PROGRAM MAIN
VAR
    sVersion: STRING:='1.0.0';
    i : UINT; //index variable for AXES()
    aFbAxes: ARRAY [1..gvl_app.axisNum] OF FB_Axis;
    hmiAxisSelection    :   INT:=1;     //Not possible to use local hmi variables for array indexes

(******Outputs: Power for Limit switches and Home Sensors (every 4th output)********)

    bOutput1 AT %Q*: BOOL:= TRUE;
    //bOutput2 AT %Q*: BOOL:= TRUE;
    //bOutput3 AT %Q*: BOOL:= TRUE;
    //bOutput4 AT %Q*: BOOL:= TRUE;
    //bOutput5 AT %Q*: BOOL:= TRUE;
    //bOutput6 AT %Q*: BOOL:= TRUE;
    //bOutput7 AT %Q*: BOOL:= TRUE;
    //bOutput8 AT %Q*: BOOL:= TRUE;
    //bOutput9 AT %Q*: BOOL:= TRUE;
    //bOutput13 AT %Q*: BOOL:= TRUE;
    //bOutput17 AT %Q*: BOOL:= TRUE;
    //bOutput21 AT %Q*: BOOL:= TRUE;
    //bOutput24 AT %Q*: BOOL:= TRUE;
    //bOutput28 AT %Q*: BOOL:= TRUE;

(******Error Handling********)
    fbErrorSystem: FB_ErrorSystem;
    aFbAxesError: ARRAY [1..gvl_app.axisNum] OF FB_NC_Error;

    //fbEL1018  : EL1018;
    //fbEL2808  : EL2808;
    //fbEL5101  : EL5101;
    //fbEL9505  : EL9505;
    //fbEL1252  : EL1252;
    //fbEL9410  : EL9410;
    //fbEL7037  : EL7037;
    //fbEK1110  : EK1110;

(******Startup, Shutdown and UPS********)
    fbUPS                  : FB_S_UPS_CX51x0;
    eUpsMode               : E_S_UPS_Mode   := eSUPS_WrPersistData_Shutdown;
    eStartUp: (ColdStart, ReadAxisFeedbackType, CheckReadDone, ExecuteRestore, CheckRestore, FinishRestore);
    bPositionRestoreDone   : BOOL := FALSE;
    bRestoreExecute        : BOOL := FALSE;
    bExecuteReadEncRefSys  : BOOL := FALSE;
    iRetry                 : INT;
    fbReadEncRefSys        : ARRAY [1..gvl_app.axisNum] OF MC_ReadParameter;
    fbRestorePosition      : ARRAY [1..GVL_app.axisNum] OF MC_SetPosition;

END_VAR

VAR PERSISTENT
    bRestoreOnStartup : BOOL;
END_VAR

fbUPS(eUpsMode := eUpsMode); (* call UPS-FB instance in first lines of the fastest PLC Task *)

IF eGlobalSUpsState = eSUPS_PowerFailure THEN
    (* first cycle of powerfailure *)
    (* execute code that should only be done once with each powerfailure, i.e. increase powerfailure counter *)
    bRestoreOnStartup:=TRUE;
    STORE_PERSISTENT();
    RETURN;
ELSIF eGlobalSUpsState > eSUPS_PowerFailure THEN
    (* next cycles of powerfailure *)
    (* skip regular code execution for the remaining cycles of the powerfailure/writing of persistent data/quick shutdown  ... *)
    RETURN;
END_IF

RESTORE_POSITIONS();
PROG();
AXES();
ERROR();

ACTION AXES:
FOR GVL.iAxis:=1 TO gvl_app.axisNum DO
    aFbAxes[GVL.iAxis](stAxisStruct:=gvl.axes[GVL.iAxis]);
END_FOR
END_ACTION

ACTION ERROR:
//
(****FB containting the log of the errors****)
//
fbErrorSystem(
    En:= TRUE,
    bReset:= ,
    nErrorNum:= ,
    bACK:= ,
    bValidSelection:= ,
    nTableRowIndex:= ,
    EnO=> ,
    nSelectedError=> ,
    pErrorSystem=> );


FOR GVL.iAxis:=1 TO gvl_app.axisNum DO
    aFbAxesError[gvl.iAxis](EN:=TRUE,
    nNC_ErrorID:= gvl.axes[gvl.iAxis].status.nErrorID,
    nNC_AxisID:=gvl.axes[gvl.iAxis].Axis.NcToPlc.AxisId,
    ErrorSystem:= fbErrorSystem.pErrorSystem);
END_FOR



(*call all the necessary instance (input assistance F2 or right click) according to the terminals that you have in your hardware and
 add "TRUE" in the input En, the corresponding number of termianl to the iTerminal_ID and
the variable "fbErrorSystem.pErrorSystem" to the input ErrorSystem in each FB E. g. :
fbEL1808(
    En:= TRUE,
    iTerminal_ID:= 01,
    ErrorSystem:= fbErorSystem.pErrorSystem,
    EnO=> ,
    bError=> );
 *)
END_ACTION

ACTION PROG:
//
(* Program any sequence, safety or feature (if necessary) application specific in thsi section*)

//
END_ACTION

ACTION RESTORE_POSITIONS:
///#########################################################
// This ACT will restore the position of an incremental axis on startup with the act position it read before losing power.
// It checks the type of axis, 0=incremental, and that the axis was stationary at shut down.
// Because 0 equates to incremental we also need to check that the data is valid, otherwise by default it would restore all axes.
// By default an axis will not restore the position unless it is set to opt-in, i.e. gvl.axes[i].config.eRestorePosition is non-zero.
// This needs to be initialised somewhere in TwinCAT code otherwise it will not be available at start up.
// A restore will only be performed on a loss of power, this code shouldn't make any changes on a reset cold, a rest origin or a download.
// There is a enum to allow for different types of restore modes, currently only one is implemented.
// 0 'DontRestore'
// 1 'RestoreWithoutHome' -restores the position using a set position fb and does not set the home bit in the axis struct.
// Note from Beckhoff: "A maximum of 1 MB persistent data can be reliably saved over the entire service life."
///#########################################################

IF bRestoreOnStartup THEN
    bRestoreOnStartup:=FALSE;
    bRestoreExecute:=TRUE;
END_IF

// Upon startup bPositionRestoreDone will be set to FALSE, after successfully completing the following code it will be set TRUE
// and should stay TRUE for the rest of the time the PLC is operational, thus this routine should only be completed once.
IF bRestoreExecute AND NOT bPositionRestoreDone THEN

    // Cycle through function blocks that read the encoder reference system i.e. whether axis is incremental or absolute
    // Result stored in Value, 0=Inc 1=Abs, execute set during the case statement
    FOR i:=1 TO gvl_app.axisNum DO
        fbReadEncRefSys[i](
          Axis:= gvl.axes[i].Axis,
          Enable:= bExecuteReadEncRefSys,
          ParameterNumber:= MC_AxisParameter.AxisEncoderReferenceSystem,
          Value=>,
          ReadMode:= E_READMODE.READMODE_ONCE);
    END_FOR

    // Cycle through set position function blocks for each axis
    FOR i:=1 TO gvl_app.axisNum DO
        fbRestorePosition[i](
         Axis:= gvl.axes[i].Axis,
         Execute:= ,
         Position:= axesPersistent[i].iPositionAtShutdown);
    END_FOR

    CASE eStartUp OF
        ColdStart:
        // First cycle of the PLC, do nothing just give one cycle for variables to initialise
            IF NOT bPositionRestoreDone THEN
                eStartUp:=eStartUp+1;
                iRetry:=0;
            END_IF

        ReadAxisFeedbackType:
        // Exectute the function blocks to read the encoder reference system (0=inc OR 1=ABS)
            bExecuteReadEncRefSys:=TRUE;
            eStartUp:=eStartUp+1;

        CheckReadDone:
        // Check the encoder reference system has been read for all axis -> if busy then continue with PLC cycle and check again next time.
        // If fbReadEncRefSys not started then go back a step.
        // If any axes result in an error the code will get stuck here, this happens if gvl_app.axisNum is not set correctly
            FOR i:=1 TO gvl_app.axisNum DO
                IF fbReadEncRefSys[i].Valid = FALSE THEN
                    IF fbReadEncRefSys[i].Busy = TRUE THEN
                        // Exit MAIN.STARTUP Action and wait till next cycle, needs to cycle through whole program in order for data to update
                        RETURN;
                    ELSE
                        // Sometimes the code gets here and the fbReadEncRefSys[i] misses the rising edge. If  the code gets here it means
                        // .valid=FALSE and .busy=FALSE which indicateds the FB probably hasn't started and thus needs to see a rising edge.
                        // Set execute to low, Exit MAIN.STARTUP and go back a step in the CASE statement.
                        bExecuteReadEncRefSys:=FALSE;
                        eStartUp:=eStartUp-1;
                        iRetry:=iRetry+1; // counter used for troubleshooting to see how many cycles it takes before fbReadEncRefSys function blocks are read correctly
                        RETURN;
                    END_IF
                END_IF
            END_FOR
            // If the code gets here all axes either have .valid=TRUE for all axes
            eStartUp:=eStartUp+1;

        ExecuteRestore:
        // Execute position restore by setting fbRestorePosition.execute = TRUE
            FOR i:=1 TO gvl_app.axisNum DO
                IF fbReadEncRefSys[i].Valid = TRUE AND fbReadEncRefSys[i].Value = 0 AND NOT(axesPersistent[i].bMovingAtShutdown) THEN
                    IF GVL.axes[i].config.eRestorePosition = RestorePosition.RestoreWithoutHome THEN
                        fbRestorePosition[i].Execute:=TRUE;
                    END_IF
                END_IF
            END_FOR
            eStartUp:=eStartUp+1;

        CheckRestore:
        // Check the set position fbs are finished
        // Nothing actually happens if the restore is not done, the code just returns from here each cycle and the
        // bPositionRestoreDone will never get set to TRUE and will take up cycle time
            FOR i:=1 TO gvl_app.axisNum DO
                IF fbReadEncRefSys[i].Valid = TRUE AND fbReadEncRefSys[i].Value = 0 AND NOT(axesPersistent[i].bMovingAtShutdown) THEN
                    IF GVL.axes[i].config.eRestorePosition = RestorePosition.RestoreWithoutHome THEN
                        IF NOT fbRestorePosition[i].Done THEN
                            RETURN;
                        END_IF
                    END_IF
                END_IF
            END_FOR
            eStartUp:=eStartUp+1;

        FinishRestore:
        // Remove execute = TRUE for fbRestorePosition
            FOR i:=1 TO gvl_app.axisNum DO
                fbRestorePosition[i].Execute:=FALSE;
            END_FOR
            bPositionRestoreDone:=TRUE;
            bRestoreExecute:=FALSE;
    END_CASE
END_IF
END_ACTION

ACTION STORE_PERSISTENT:
FOR i:=1 TO gvl_app.axisNum DO
    axesPersistent[i].iPositionAtShutdown:=gvl.axes[i].Axis.NcToPlc.ActPos;
    IF gvl.axes[i].Axis.NcToPlc.ActVelo <> 0 THEN
        axesPersistent[i].bMovingAtShutdown:=TRUE;
    ELSE
        axesPersistent[i].bMovingAtShutdown:=FALSE;
    END_IF
    axesPersistent[i].bMovingAtShutdown:=axesPersistent[i].bMovingAtShutdown OR gvl.axes[i].Axis.Status.Moving;
END_FOR
END_ACTION

END_PROGRAM

(* stored: Version 1.1.0.1, ProductVersion 3.1.4024.0
   POU MAIN: Id {33eb6f49-7781-4211-a70b-87ada6d80cb7}, SpecialFunc None
   Action AXES: Id {7eb32732-9b53-4934-8cd9-20ba971dd8ff}
   Action ERROR: Id {35f2cf38-f81e-4aa3-9534-be5fb417817d}
   Action PROG: Id {5d03ebbb-2a47-4890-ad6d-e82daf72dc51}
   Action RESTORE_POSITIONS: Id {0c7ee537-7bd9-4833-b428-c17cbb57e893}
   Action STORE_PERSISTENT: Id {cb5c9254-2e5f-47b1-9baa-10e728a961b0} *)
